PROPERTY bogKeyFilterOverloadToolValue : BOOL
GET
                    bogKeyFilterOverloadToolValue := bogKeyFilterOverload.Value;

                  
END_GET
SET
                    bogKeyFilterOverload.Value := bogKeyFilterOverloadToolValue;

                  
END_SET
END_PROPERTY

PROPERTY bogKeyNextModeToolValue : BOOL
GET
                    bogKeyNextModeToolValue := bogKeyNextMode.Value;

                  
END_GET
SET
                    bogKeyNextMode.Value := bogKeyNextModeToolValue;

                  
END_SET
END_PROPERTY

PROPERTY bogKeyPrevModeToolValue : BOOL
GET
                    bogKeyPrevModeToolValue := bogKeyPrevMode.Value;

                  
END_GET
SET
                    bogKeyPrevMode.Value := bogKeyPrevModeToolValue;

                  
END_SET
END_PROPERTY

PROPERTY bogKeySignalDangerToolValue : BOOL
GET
                    bogKeySignalDangerToolValue := bogKeySignalDanger.Value;

                  
END_GET
SET
                    bogKeySignalDanger.Value := bogKeySignalDangerToolValue;

                  
END_SET
END_PROPERTY

PROPERTY bogKeyFlashLightONToolValue : BOOL
GET
                    bogKeyFlashLightONToolValue := bogKeyFlashLightON.Value;

                  
END_GET
SET
                    bogKeyFlashLightON.Value := bogKeyFlashLightONToolValue;

                  
END_SET
END_PROPERTY

PROPERTY bogKeyCalibMastMinToolValue : BOOL
GET
                    bogKeyCalibMastMinToolValue := bogKeyCalibMastMin.Value;

                  
END_GET
SET
                    bogKeyCalibMastMin.Value := bogKeyCalibMastMinToolValue;

                  
END_SET
END_PROPERTY

PROPERTY bogKeyCalibMastMaxToolValue : BOOL
GET
                    bogKeyCalibMastMaxToolValue := bogKeyCalibMastMax.Value;

                  
END_GET
SET
                    bogKeyCalibMastMax.Value := bogKeyCalibMastMaxToolValue;

                  
END_SET
END_PROPERTY

PROPERTY bogKeyCalibMastValidToolValue : BOOL
GET
                    bogKeyCalibMastValidToolValue := bogKeyCalibMastValid.Value;

                  
END_GET
SET
                    bogKeyCalibMastValid.Value := bogKeyCalibMastValidToolValue;

                  
END_SET
END_PROPERTY

PROPERTY bogKeyGeneratorActivateToolValue : BOOL
GET
                    bogKeyGeneratorActivateToolValue := bogKeyGeneratorActivate.Value;

                  
END_GET
SET
                    bogKeyGeneratorActivate.Value := bogKeyGeneratorActivateToolValue;

                  
END_SET
END_PROPERTY

PROPERTY bogKeyWhiteLights15746ToolValue : BOOL
GET
                    bogKeyWhiteLights15746ToolValue := bogKeyWhiteLights15746.Value;

                  
END_GET
SET
                    bogKeyWhiteLights15746.Value := bogKeyWhiteLights15746ToolValue;

                  
END_SET
END_PROPERTY

PROPERTY bogFixe2ndParkBrakeSelectToolValue : BOOL
GET
                    bogFixe2ndParkBrakeSelectToolValue := bogFixe2ndParkBrakeSelect.Value;

                  
END_GET
SET
                    bogFixe2ndParkBrakeSelect.Value := bogFixe2ndParkBrakeSelectToolValue;

                  
END_SET
END_PROPERTY

PROPERTY bogOsci2ndParkBrakeSelectToolValue : BOOL
GET
                    bogOsci2ndParkBrakeSelectToolValue := bogOsci2ndParkBrakeSelect.Value;

                  
END_GET
SET
                    bogOsci2ndParkBrakeSelect.Value := bogOsci2ndParkBrakeSelectToolValue;

                  
END_SET
END_PROPERTY

PROPERTY bogKeyRazControllerToolValue : BOOL
GET
                    bogKeyRazControllerToolValue := bogKeyRazController.Value;

                  
END_GET
SET
                    bogKeyRazController.Value := bogKeyRazControllerToolValue;

                  
END_SET
END_PROPERTY

METHOD InitializeCanSignals
                  bogLoginStatus.AppScalingDivisor :=1;
bogLoginStatus.AppScalingMultiplier :=1;
bogLoginStatus.AppScalingOffset :=0;
bogLoginStatus.AppUnit :="[-]";
bogLoginStatus.CanDefault :=0;
bogLoginStatus.CanInit :=0;
bogLoginStatus.CanMax :=1;
bogLoginStatus.CanMin :=0;
bogLoginStatus.CanUnit :="";
bogLoginStatus.Description :="User Log in Status (1=log in)";
bogLoginStatus.ErrorReaction := eErrorReaction.ERSIG_DFLT;
bogLoginStatus.ReceiverAdress :=1;
bogLoginStatus.ToolScalingDivisor :=1;
bogLoginStatus.ToolScalingMultiplier :=1;
bogLoginStatus.ToolScalingOffset :=0;
bogLoginStatus.ToolUnit :="";

bogButtonCalibTurretEncoder.AppScalingDivisor :=1;
bogButtonCalibTurretEncoder.AppScalingMultiplier :=1;
bogButtonCalibTurretEncoder.AppScalingOffset :=0;
bogButtonCalibTurretEncoder.AppUnit :="[-]";
bogButtonCalibTurretEncoder.CanDefault :=0;
bogButtonCalibTurretEncoder.CanInit :=0;
bogButtonCalibTurretEncoder.CanMax :=1;
bogButtonCalibTurretEncoder.CanMin :=0;
bogButtonCalibTurretEncoder.CanUnit :="";
bogButtonCalibTurretEncoder.Description :="Button for the calibration of the turret encoder is pressed";
bogButtonCalibTurretEncoder.ErrorReaction := eErrorReaction.ERSIG_DFLT;
bogButtonCalibTurretEncoder.ReceiverAdress :=1;
bogButtonCalibTurretEncoder.ToolScalingDivisor :=1;
bogButtonCalibTurretEncoder.ToolScalingMultiplier :=1;
bogButtonCalibTurretEncoder.ToolScalingOffset :=0;
bogButtonCalibTurretEncoder.ToolUnit :="";

bogButtonCalibMinMastMeasure.AppScalingDivisor :=1;
bogButtonCalibMinMastMeasure.AppScalingMultiplier :=1;
bogButtonCalibMinMastMeasure.AppScalingOffset :=0;
bogButtonCalibMinMastMeasure.AppUnit :="[-]";
bogButtonCalibMinMastMeasure.CanDefault :=0;
bogButtonCalibMinMastMeasure.CanInit :=0;
bogButtonCalibMinMastMeasure.CanMax :=1;
bogButtonCalibMinMastMeasure.CanMin :=0;
bogButtonCalibMinMastMeasure.CanUnit :="";
bogButtonCalibMinMastMeasure.Description :="Button for the calibration of min position mast measure encodeur  is pressed";
bogButtonCalibMinMastMeasure.ErrorReaction := eErrorReaction.ERSIG_DFLT;
bogButtonCalibMinMastMeasure.ReceiverAdress :=1;
bogButtonCalibMinMastMeasure.ToolScalingDivisor :=1;
bogButtonCalibMinMastMeasure.ToolScalingMultiplier :=1;
bogButtonCalibMinMastMeasure.ToolScalingOffset :=0;
bogButtonCalibMinMastMeasure.ToolUnit :="";

bogButtonCalibMaxMastMeasure.AppScalingDivisor :=1;
bogButtonCalibMaxMastMeasure.AppScalingMultiplier :=1;
bogButtonCalibMaxMastMeasure.AppScalingOffset :=0;
bogButtonCalibMaxMastMeasure.AppUnit :="[-]";
bogButtonCalibMaxMastMeasure.CanDefault :=0;
bogButtonCalibMaxMastMeasure.CanInit :=0;
bogButtonCalibMaxMastMeasure.CanMax :=1;
bogButtonCalibMaxMastMeasure.CanMin :=0;
bogButtonCalibMaxMastMeasure.CanUnit :="";
bogButtonCalibMaxMastMeasure.Description :="Button for the calibration of max position mast measure encodeur  is pressed";
bogButtonCalibMaxMastMeasure.ErrorReaction := eErrorReaction.ERSIG_DFLT;
bogButtonCalibMaxMastMeasure.ReceiverAdress :=1;
bogButtonCalibMaxMastMeasure.ToolScalingDivisor :=1;
bogButtonCalibMaxMastMeasure.ToolScalingMultiplier :=1;
bogButtonCalibMaxMastMeasure.ToolScalingOffset :=0;
bogButtonCalibMaxMastMeasure.ToolUnit :="";

boSavePosEncodeurMastButton.AppScalingDivisor :=1;
boSavePosEncodeurMastButton.AppScalingMultiplier :=1;
boSavePosEncodeurMastButton.AppScalingOffset :=0;
boSavePosEncodeurMastButton.AppUnit :="[-]";
boSavePosEncodeurMastButton.CanDefault :=0;
boSavePosEncodeurMastButton.CanInit :=0;
boSavePosEncodeurMastButton.CanMax :=1;
boSavePosEncodeurMastButton.CanMin :=0;
boSavePosEncodeurMastButton.CanUnit :="";
boSavePosEncodeurMastButton.Description :="Button for save min and max value of encodeur mast measure";
boSavePosEncodeurMastButton.ErrorReaction := eErrorReaction.ERSIG_DFLT;
boSavePosEncodeurMastButton.ReceiverAdress :=1;
boSavePosEncodeurMastButton.ToolScalingDivisor :=1;
boSavePosEncodeurMastButton.ToolScalingMultiplier :=1;
boSavePosEncodeurMastButton.ToolScalingOffset :=0;
boSavePosEncodeurMastButton.ToolUnit :="";

bogActivateMeasuringMast.AppScalingDivisor :=1;
bogActivateMeasuringMast.AppScalingMultiplier :=1;
bogActivateMeasuringMast.AppScalingOffset :=0;
bogActivateMeasuringMast.AppUnit :="[-]";
bogActivateMeasuringMast.CanDefault :=0;
bogActivateMeasuringMast.CanInit :=0;
bogActivateMeasuringMast.CanMax :=1;
bogActivateMeasuringMast.CanMin :=0;
bogActivateMeasuringMast.CanUnit :="";
bogActivateMeasuringMast.Description :="Activate mast measure function";
bogActivateMeasuringMast.ErrorReaction := eErrorReaction.ERSIG_DFLT;
bogActivateMeasuringMast.ReceiverAdress :=1;
bogActivateMeasuringMast.ToolScalingDivisor :=1;
bogActivateMeasuringMast.ToolScalingMultiplier :=1;
bogActivateMeasuringMast.ToolScalingOffset :=0;
bogActivateMeasuringMast.ToolUnit :="";

boRazDistanceTraveledMastMeasure.AppScalingDivisor :=1;
boRazDistanceTraveledMastMeasure.AppScalingMultiplier :=1;
boRazDistanceTraveledMastMeasure.AppScalingOffset :=0;
boRazDistanceTraveledMastMeasure.AppUnit :="[-]";
boRazDistanceTraveledMastMeasure.CanDefault :=0;
boRazDistanceTraveledMastMeasure.CanInit :=0;
boRazDistanceTraveledMastMeasure.CanMax :=1;
boRazDistanceTraveledMastMeasure.CanMin :=0;
boRazDistanceTraveledMastMeasure.CanUnit :="";
boRazDistanceTraveledMastMeasure.Description :="Raz distance translation traveled with mast measure unfolded";
boRazDistanceTraveledMastMeasure.ErrorReaction := eErrorReaction.ERSIG_DFLT;
boRazDistanceTraveledMastMeasure.ReceiverAdress :=1;
boRazDistanceTraveledMastMeasure.ToolScalingDivisor :=1;
boRazDistanceTraveledMastMeasure.ToolScalingMultiplier :=1;
boRazDistanceTraveledMastMeasure.ToolScalingOffset :=0;
boRazDistanceTraveledMastMeasure.ToolUnit :="";

bogOffTrackTestBrakeActivated.AppScalingDivisor :=1;
bogOffTrackTestBrakeActivated.AppScalingMultiplier :=1;
bogOffTrackTestBrakeActivated.AppScalingOffset :=0;
bogOffTrackTestBrakeActivated.AppUnit :="[-]";
bogOffTrackTestBrakeActivated.CanDefault :=0;
bogOffTrackTestBrakeActivated.CanInit :=0;
bogOffTrackTestBrakeActivated.CanMax :=1;
bogOffTrackTestBrakeActivated.CanMin :=0;
bogOffTrackTestBrakeActivated.CanUnit :="";
bogOffTrackTestBrakeActivated.Description :="Status of off track variable on test brake page";
bogOffTrackTestBrakeActivated.ErrorReaction := eErrorReaction.ERSIG_DFLT;
bogOffTrackTestBrakeActivated.ReceiverAdress :=1;
bogOffTrackTestBrakeActivated.ToolScalingDivisor :=1;
bogOffTrackTestBrakeActivated.ToolScalingMultiplier :=1;
bogOffTrackTestBrakeActivated.ToolScalingOffset :=0;
bogOffTrackTestBrakeActivated.ToolUnit :="";

bogOffTrackRunInBrakeActivated.AppScalingDivisor :=1;
bogOffTrackRunInBrakeActivated.AppScalingMultiplier :=1;
bogOffTrackRunInBrakeActivated.AppScalingOffset :=0;
bogOffTrackRunInBrakeActivated.AppUnit :="[-]";
bogOffTrackRunInBrakeActivated.CanDefault :=0;
bogOffTrackRunInBrakeActivated.CanInit :=0;
bogOffTrackRunInBrakeActivated.CanMax :=1;
bogOffTrackRunInBrakeActivated.CanMin :=0;
bogOffTrackRunInBrakeActivated.CanUnit :="";
bogOffTrackRunInBrakeActivated.Description :="Status of off track variable on run in process page";
bogOffTrackRunInBrakeActivated.ErrorReaction := eErrorReaction.ERSIG_DFLT;
bogOffTrackRunInBrakeActivated.ReceiverAdress :=1;
bogOffTrackRunInBrakeActivated.ToolScalingDivisor :=1;
bogOffTrackRunInBrakeActivated.ToolScalingMultiplier :=1;
bogOffTrackRunInBrakeActivated.ToolScalingOffset :=0;
bogOffTrackRunInBrakeActivated.ToolUnit :="";

bogOsciServiceBrakeSelect.AppScalingDivisor :=1;
bogOsciServiceBrakeSelect.AppScalingMultiplier :=1;
bogOsciServiceBrakeSelect.AppScalingOffset :=0;
bogOsciServiceBrakeSelect.AppUnit :="[-]";
bogOsciServiceBrakeSelect.CanDefault :=0;
bogOsciServiceBrakeSelect.CanInit :=0;
bogOsciServiceBrakeSelect.CanMax :=1;
bogOsciServiceBrakeSelect.CanMin :=0;
bogOsciServiceBrakeSelect.CanUnit :="";
bogOsciServiceBrakeSelect.Description :="Request status of osci service test brake";
bogOsciServiceBrakeSelect.ErrorReaction := eErrorReaction.ERSIG_DFLT;
bogOsciServiceBrakeSelect.ReceiverAdress :=1;
bogOsciServiceBrakeSelect.ToolScalingDivisor :=1;
bogOsciServiceBrakeSelect.ToolScalingMultiplier :=1;
bogOsciServiceBrakeSelect.ToolScalingOffset :=0;
bogOsciServiceBrakeSelect.ToolUnit :="";

bogFixedServiceBrakeSelect.AppScalingDivisor :=1;
bogFixedServiceBrakeSelect.AppScalingMultiplier :=1;
bogFixedServiceBrakeSelect.AppScalingOffset :=0;
bogFixedServiceBrakeSelect.AppUnit :="[-]";
bogFixedServiceBrakeSelect.CanDefault :=0;
bogFixedServiceBrakeSelect.CanInit :=0;
bogFixedServiceBrakeSelect.CanMax :=1;
bogFixedServiceBrakeSelect.CanMin :=0;
bogFixedServiceBrakeSelect.CanUnit :="";
bogFixedServiceBrakeSelect.Description :="Request status of fixed service test brake";
bogFixedServiceBrakeSelect.ErrorReaction := eErrorReaction.ERSIG_DFLT;
bogFixedServiceBrakeSelect.ReceiverAdress :=1;
bogFixedServiceBrakeSelect.ToolScalingDivisor :=1;
bogFixedServiceBrakeSelect.ToolScalingMultiplier :=1;
bogFixedServiceBrakeSelect.ToolScalingOffset :=0;
bogFixedServiceBrakeSelect.ToolUnit :="";

bogBothServiceBrakeSelect.AppScalingDivisor :=1;
bogBothServiceBrakeSelect.AppScalingMultiplier :=1;
bogBothServiceBrakeSelect.AppScalingOffset :=0;
bogBothServiceBrakeSelect.AppUnit :="[-]";
bogBothServiceBrakeSelect.CanDefault :=0;
bogBothServiceBrakeSelect.CanInit :=0;
bogBothServiceBrakeSelect.CanMax :=1;
bogBothServiceBrakeSelect.CanMin :=0;
bogBothServiceBrakeSelect.CanUnit :="";
bogBothServiceBrakeSelect.Description :="Request status of both service test brake";
bogBothServiceBrakeSelect.ErrorReaction := eErrorReaction.ERSIG_DFLT;
bogBothServiceBrakeSelect.ReceiverAdress :=1;
bogBothServiceBrakeSelect.ToolScalingDivisor :=1;
bogBothServiceBrakeSelect.ToolScalingMultiplier :=1;
bogBothServiceBrakeSelect.ToolScalingOffset :=0;
bogBothServiceBrakeSelect.ToolUnit :="";

bogOsciParkBrakeSelect.AppScalingDivisor :=1;
bogOsciParkBrakeSelect.AppScalingMultiplier :=1;
bogOsciParkBrakeSelect.AppScalingOffset :=0;
bogOsciParkBrakeSelect.AppUnit :="[-]";
bogOsciParkBrakeSelect.CanDefault :=0;
bogOsciParkBrakeSelect.CanInit :=0;
bogOsciParkBrakeSelect.CanMax :=1;
bogOsciParkBrakeSelect.CanMin :=0;
bogOsciParkBrakeSelect.CanUnit :="";
bogOsciParkBrakeSelect.Description :="Request status of osci park test brake";
bogOsciParkBrakeSelect.ErrorReaction := eErrorReaction.ERSIG_DFLT;
bogOsciParkBrakeSelect.ReceiverAdress :=1;
bogOsciParkBrakeSelect.ToolScalingDivisor :=1;
bogOsciParkBrakeSelect.ToolScalingMultiplier :=1;
bogOsciParkBrakeSelect.ToolScalingOffset :=0;
bogOsciParkBrakeSelect.ToolUnit :="";

bogFixedParkBrakeSelect.AppScalingDivisor :=1;
bogFixedParkBrakeSelect.AppScalingMultiplier :=1;
bogFixedParkBrakeSelect.AppScalingOffset :=0;
bogFixedParkBrakeSelect.AppUnit :="[-]";
bogFixedParkBrakeSelect.CanDefault :=0;
bogFixedParkBrakeSelect.CanInit :=0;
bogFixedParkBrakeSelect.CanMax :=1;
bogFixedParkBrakeSelect.CanMin :=0;
bogFixedParkBrakeSelect.CanUnit :="";
bogFixedParkBrakeSelect.Description :="Request status of fixed park test brake";
bogFixedParkBrakeSelect.ErrorReaction := eErrorReaction.ERSIG_DFLT;
bogFixedParkBrakeSelect.ReceiverAdress :=1;
bogFixedParkBrakeSelect.ToolScalingDivisor :=1;
bogFixedParkBrakeSelect.ToolScalingMultiplier :=1;
bogFixedParkBrakeSelect.ToolScalingOffset :=0;
bogFixedParkBrakeSelect.ToolUnit :="";

bogBothParkBrakeSelect.AppScalingDivisor :=1;
bogBothParkBrakeSelect.AppScalingMultiplier :=1;
bogBothParkBrakeSelect.AppScalingOffset :=0;
bogBothParkBrakeSelect.AppUnit :="[-]";
bogBothParkBrakeSelect.CanDefault :=0;
bogBothParkBrakeSelect.CanInit :=0;
bogBothParkBrakeSelect.CanMax :=1;
bogBothParkBrakeSelect.CanMin :=0;
bogBothParkBrakeSelect.CanUnit :="";
bogBothParkBrakeSelect.Description :="Request status of both park test brake";
bogBothParkBrakeSelect.ErrorReaction := eErrorReaction.ERSIG_DFLT;
bogBothParkBrakeSelect.ReceiverAdress :=1;
bogBothParkBrakeSelect.ToolScalingDivisor :=1;
bogBothParkBrakeSelect.ToolScalingMultiplier :=1;
bogBothParkBrakeSelect.ToolScalingOffset :=0;
bogBothParkBrakeSelect.ToolUnit :="";

bogOsciServiceRunInBrakeSelect.AppScalingDivisor :=1;
bogOsciServiceRunInBrakeSelect.AppScalingMultiplier :=1;
bogOsciServiceRunInBrakeSelect.AppScalingOffset :=0;
bogOsciServiceRunInBrakeSelect.AppUnit :="[-]";
bogOsciServiceRunInBrakeSelect.CanDefault :=0;
bogOsciServiceRunInBrakeSelect.CanInit :=0;
bogOsciServiceRunInBrakeSelect.CanMax :=1;
bogOsciServiceRunInBrakeSelect.CanMin :=0;
bogOsciServiceRunInBrakeSelect.CanUnit :="";
bogOsciServiceRunInBrakeSelect.Description :="Request status of osci service run in brake";
bogOsciServiceRunInBrakeSelect.ErrorReaction := eErrorReaction.ERSIG_DFLT;
bogOsciServiceRunInBrakeSelect.ReceiverAdress :=1;
bogOsciServiceRunInBrakeSelect.ToolScalingDivisor :=1;
bogOsciServiceRunInBrakeSelect.ToolScalingMultiplier :=1;
bogOsciServiceRunInBrakeSelect.ToolScalingOffset :=0;
bogOsciServiceRunInBrakeSelect.ToolUnit :="";

bogFixedServiceRunInBrakeSelect.AppScalingDivisor :=1;
bogFixedServiceRunInBrakeSelect.AppScalingMultiplier :=1;
bogFixedServiceRunInBrakeSelect.AppScalingOffset :=0;
bogFixedServiceRunInBrakeSelect.AppUnit :="[-]";
bogFixedServiceRunInBrakeSelect.CanDefault :=0;
bogFixedServiceRunInBrakeSelect.CanInit :=0;
bogFixedServiceRunInBrakeSelect.CanMax :=1;
bogFixedServiceRunInBrakeSelect.CanMin :=0;
bogFixedServiceRunInBrakeSelect.CanUnit :="";
bogFixedServiceRunInBrakeSelect.Description :="Request status of fixed service run in test brake";
bogFixedServiceRunInBrakeSelect.ErrorReaction := eErrorReaction.ERSIG_DFLT;
bogFixedServiceRunInBrakeSelect.ReceiverAdress :=1;
bogFixedServiceRunInBrakeSelect.ToolScalingDivisor :=1;
bogFixedServiceRunInBrakeSelect.ToolScalingMultiplier :=1;
bogFixedServiceRunInBrakeSelect.ToolScalingOffset :=0;
bogFixedServiceRunInBrakeSelect.ToolUnit :="";

bogBothServiceRunInBrakeSelect.AppScalingDivisor :=1;
bogBothServiceRunInBrakeSelect.AppScalingMultiplier :=1;
bogBothServiceRunInBrakeSelect.AppScalingOffset :=0;
bogBothServiceRunInBrakeSelect.AppUnit :="[-]";
bogBothServiceRunInBrakeSelect.CanDefault :=0;
bogBothServiceRunInBrakeSelect.CanInit :=0;
bogBothServiceRunInBrakeSelect.CanMax :=1;
bogBothServiceRunInBrakeSelect.CanMin :=0;
bogBothServiceRunInBrakeSelect.CanUnit :="";
bogBothServiceRunInBrakeSelect.Description :="Request status of both service run in test brake";
bogBothServiceRunInBrakeSelect.ErrorReaction := eErrorReaction.ERSIG_DFLT;
bogBothServiceRunInBrakeSelect.ReceiverAdress :=1;
bogBothServiceRunInBrakeSelect.ToolScalingDivisor :=1;
bogBothServiceRunInBrakeSelect.ToolScalingMultiplier :=1;
bogBothServiceRunInBrakeSelect.ToolScalingOffset :=0;
bogBothServiceRunInBrakeSelect.ToolUnit :="";

bogTestBrakePageActive.AppScalingDivisor :=1;
bogTestBrakePageActive.AppScalingMultiplier :=1;
bogTestBrakePageActive.AppScalingOffset :=0;
bogTestBrakePageActive.AppUnit :="[-]";
bogTestBrakePageActive.CanDefault :=0;
bogTestBrakePageActive.CanInit :=0;
bogTestBrakePageActive.CanMax :=1;
bogTestBrakePageActive.CanMin :=0;
bogTestBrakePageActive.CanUnit :="";
bogTestBrakePageActive.Description :="Flag when user is on test brake page";
bogTestBrakePageActive.ErrorReaction := eErrorReaction.ERSIG_DFLT;
bogTestBrakePageActive.ReceiverAdress :=1;
bogTestBrakePageActive.ToolScalingDivisor :=1;
bogTestBrakePageActive.ToolScalingMultiplier :=1;
bogTestBrakePageActive.ToolScalingOffset :=0;
bogTestBrakePageActive.ToolUnit :="";

bogBreakInBrakePageActive.AppScalingDivisor :=1;
bogBreakInBrakePageActive.AppScalingMultiplier :=1;
bogBreakInBrakePageActive.AppScalingOffset :=0;
bogBreakInBrakePageActive.AppUnit :="[-]";
bogBreakInBrakePageActive.CanDefault :=0;
bogBreakInBrakePageActive.CanInit :=0;
bogBreakInBrakePageActive.CanMax :=1;
bogBreakInBrakePageActive.CanMin :=0;
bogBreakInBrakePageActive.CanUnit :="";
bogBreakInBrakePageActive.Description :="Flag when user is on break in brake page";
bogBreakInBrakePageActive.ErrorReaction := eErrorReaction.ERSIG_DFLT;
bogBreakInBrakePageActive.ReceiverAdress :=1;
bogBreakInBrakePageActive.ToolScalingDivisor :=1;
bogBreakInBrakePageActive.ToolScalingMultiplier :=1;
bogBreakInBrakePageActive.ToolScalingOffset :=0;
bogBreakInBrakePageActive.ToolUnit :="";

bogSerialNumber.AppScalingDivisor :=1;
bogSerialNumber.AppScalingMultiplier :=1;
bogSerialNumber.AppScalingOffset :=0;
bogSerialNumber.AppUnit :="[-]";
bogSerialNumber.CanDefault :=0;
bogSerialNumber.CanInit :=0;
bogSerialNumber.CanMax :=1;
bogSerialNumber.CanMin :=0;
bogSerialNumber.CanUnit :="";
bogSerialNumber.Description :="Machine Serial Number";
bogSerialNumber.ErrorReaction := eErrorReaction.ERSIG_DFLT;
bogSerialNumber.ReceiverAdress :=1;
bogSerialNumber.ToolScalingDivisor :=1;
bogSerialNumber.ToolScalingMultiplier :=1;
bogSerialNumber.ToolScalingOffset :=0;
bogSerialNumber.ToolUnit :="";

bogBPBasketValidate.AppScalingDivisor :=1;
bogBPBasketValidate.AppScalingMultiplier :=1;
bogBPBasketValidate.AppScalingOffset :=0;
bogBPBasketValidate.AppUnit :="[-]";
bogBPBasketValidate.CanDefault :=0;
bogBPBasketValidate.CanInit :=0;
bogBPBasketValidate.CanMax :=1;
bogBPBasketValidate.CanMin :=0;
bogBPBasketValidate.CanUnit :="";
bogBPBasketValidate.Description :="Basket Panel Validate";
bogBPBasketValidate.ErrorReaction := eErrorReaction.ERSIG_DFLT;
bogBPBasketValidate.ReceiverAdress :=1;
bogBPBasketValidate.ToolScalingDivisor :=1;
bogBPBasketValidate.ToolScalingMultiplier :=1;
bogBPBasketValidate.ToolScalingOffset :=0;
bogBPBasketValidate.ToolUnit :="";

bogKeyFilterOverload.AppScalingDivisor :=1;
bogKeyFilterOverload.AppScalingMultiplier :=1;
bogKeyFilterOverload.AppScalingOffset :=0;
bogKeyFilterOverload.AppUnit :="[-]";
bogKeyFilterOverload.CanDefault :=0;
bogKeyFilterOverload.CanInit :=0;
bogKeyFilterOverload.CanMax :=1;
bogKeyFilterOverload.CanMin :=0;
bogKeyFilterOverload.CanUnit :="";
bogKeyFilterOverload.Description :="Overload Filter Key";
bogKeyFilterOverload.ErrorReaction := eErrorReaction.ERSIG_DFLT;
bogKeyFilterOverload.ReceiverAdress :=1;
bogKeyFilterOverload.ToolScalingDivisor :=1;
bogKeyFilterOverload.ToolScalingMultiplier :=1;
bogKeyFilterOverload.ToolScalingOffset :=0;
bogKeyFilterOverload.ToolUnit :="";

bogKeyNextMode.AppScalingDivisor :=1;
bogKeyNextMode.AppScalingMultiplier :=1;
bogKeyNextMode.AppScalingOffset :=0;
bogKeyNextMode.AppUnit :="[-]";
bogKeyNextMode.CanDefault :=0;
bogKeyNextMode.CanInit :=0;
bogKeyNextMode.CanMax :=1;
bogKeyNextMode.CanMin :=0;
bogKeyNextMode.CanUnit :="";
bogKeyNextMode.Description :="Select next mode";
bogKeyNextMode.ErrorReaction := eErrorReaction.ERSIG_DFLT;
bogKeyNextMode.ReceiverAdress :=1;
bogKeyNextMode.ToolScalingDivisor :=1;
bogKeyNextMode.ToolScalingMultiplier :=1;
bogKeyNextMode.ToolScalingOffset :=0;
bogKeyNextMode.ToolUnit :="";

bogKeyPrevMode.AppScalingDivisor :=1;
bogKeyPrevMode.AppScalingMultiplier :=1;
bogKeyPrevMode.AppScalingOffset :=0;
bogKeyPrevMode.AppUnit :="[-]";
bogKeyPrevMode.CanDefault :=0;
bogKeyPrevMode.CanInit :=0;
bogKeyPrevMode.CanMax :=1;
bogKeyPrevMode.CanMin :=0;
bogKeyPrevMode.CanUnit :="";
bogKeyPrevMode.Description :="Select Previous Mode";
bogKeyPrevMode.ErrorReaction := eErrorReaction.ERSIG_DFLT;
bogKeyPrevMode.ReceiverAdress :=1;
bogKeyPrevMode.ToolScalingDivisor :=1;
bogKeyPrevMode.ToolScalingMultiplier :=1;
bogKeyPrevMode.ToolScalingOffset :=0;
bogKeyPrevMode.ToolUnit :="";

bogKeySignalDanger.AppScalingDivisor :=1;
bogKeySignalDanger.AppScalingMultiplier :=1;
bogKeySignalDanger.AppScalingOffset :=0;
bogKeySignalDanger.AppUnit :="[-]";
bogKeySignalDanger.CanDefault :=0;
bogKeySignalDanger.CanInit :=0;
bogKeySignalDanger.CanMax :=1;
bogKeySignalDanger.CanMin :=0;
bogKeySignalDanger.CanUnit :="";
bogKeySignalDanger.Description :="Select Signal Danger Mode";
bogKeySignalDanger.ErrorReaction := eErrorReaction.ERSIG_DFLT;
bogKeySignalDanger.ReceiverAdress :=1;
bogKeySignalDanger.ToolScalingDivisor :=1;
bogKeySignalDanger.ToolScalingMultiplier :=1;
bogKeySignalDanger.ToolScalingOffset :=0;
bogKeySignalDanger.ToolUnit :="";

bogKeyFlashLightON.AppScalingDivisor :=1;
bogKeyFlashLightON.AppScalingMultiplier :=1;
bogKeyFlashLightON.AppScalingOffset :=0;
bogKeyFlashLightON.AppUnit :="[-]";
bogKeyFlashLightON.CanDefault :=0;
bogKeyFlashLightON.CanInit :=0;
bogKeyFlashLightON.CanMax :=1;
bogKeyFlashLightON.CanMin :=0;
bogKeyFlashLightON.CanUnit :="";
bogKeyFlashLightON.Description :="Force Flash Light ON";
bogKeyFlashLightON.ErrorReaction := eErrorReaction.ERSIG_DFLT;
bogKeyFlashLightON.ReceiverAdress :=1;
bogKeyFlashLightON.ToolScalingDivisor :=1;
bogKeyFlashLightON.ToolScalingMultiplier :=1;
bogKeyFlashLightON.ToolScalingOffset :=0;
bogKeyFlashLightON.ToolUnit :="";

bogKeyCalibMastMin.AppScalingDivisor :=1;
bogKeyCalibMastMin.AppScalingMultiplier :=1;
bogKeyCalibMastMin.AppScalingOffset :=0;
bogKeyCalibMastMin.AppUnit :="[-]";
bogKeyCalibMastMin.CanDefault :=0;
bogKeyCalibMastMin.CanInit :=0;
bogKeyCalibMastMin.CanMax :=1;
bogKeyCalibMastMin.CanMin :=0;
bogKeyCalibMastMin.CanUnit :="";
bogKeyCalibMastMin.Description :="Key Calibration Min";
bogKeyCalibMastMin.ErrorReaction := eErrorReaction.ERSIG_DFLT;
bogKeyCalibMastMin.ReceiverAdress :=1;
bogKeyCalibMastMin.ToolScalingDivisor :=1;
bogKeyCalibMastMin.ToolScalingMultiplier :=1;
bogKeyCalibMastMin.ToolScalingOffset :=0;
bogKeyCalibMastMin.ToolUnit :="";

bogKeyCalibMastMax.AppScalingDivisor :=1;
bogKeyCalibMastMax.AppScalingMultiplier :=1;
bogKeyCalibMastMax.AppScalingOffset :=0;
bogKeyCalibMastMax.AppUnit :="[-]";
bogKeyCalibMastMax.CanDefault :=0;
bogKeyCalibMastMax.CanInit :=0;
bogKeyCalibMastMax.CanMax :=1;
bogKeyCalibMastMax.CanMin :=0;
bogKeyCalibMastMax.CanUnit :="";
bogKeyCalibMastMax.Description :="Key Calibration Max";
bogKeyCalibMastMax.ErrorReaction := eErrorReaction.ERSIG_DFLT;
bogKeyCalibMastMax.ReceiverAdress :=1;
bogKeyCalibMastMax.ToolScalingDivisor :=1;
bogKeyCalibMastMax.ToolScalingMultiplier :=1;
bogKeyCalibMastMax.ToolScalingOffset :=0;
bogKeyCalibMastMax.ToolUnit :="";

bogKeyCalibMastValid.AppScalingDivisor :=1;
bogKeyCalibMastValid.AppScalingMultiplier :=1;
bogKeyCalibMastValid.AppScalingOffset :=0;
bogKeyCalibMastValid.AppUnit :="[-]";
bogKeyCalibMastValid.CanDefault :=0;
bogKeyCalibMastValid.CanInit :=0;
bogKeyCalibMastValid.CanMax :=1;
bogKeyCalibMastValid.CanMin :=0;
bogKeyCalibMastValid.CanUnit :="";
bogKeyCalibMastValid.Description :="Key Calibration Validation";
bogKeyCalibMastValid.ErrorReaction := eErrorReaction.ERSIG_DFLT;
bogKeyCalibMastValid.ReceiverAdress :=1;
bogKeyCalibMastValid.ToolScalingDivisor :=1;
bogKeyCalibMastValid.ToolScalingMultiplier :=1;
bogKeyCalibMastValid.ToolScalingOffset :=0;
bogKeyCalibMastValid.ToolUnit :="";

bogKeyGeneratorActivate.AppScalingDivisor :=1;
bogKeyGeneratorActivate.AppScalingMultiplier :=1;
bogKeyGeneratorActivate.AppScalingOffset :=0;
bogKeyGeneratorActivate.AppUnit :="[-]";
bogKeyGeneratorActivate.CanDefault :=0;
bogKeyGeneratorActivate.CanInit :=0;
bogKeyGeneratorActivate.CanMax :=1;
bogKeyGeneratorActivate.CanMin :=0;
bogKeyGeneratorActivate.CanUnit :="";
bogKeyGeneratorActivate.Description :="Key Generator Activation";
bogKeyGeneratorActivate.ErrorReaction := eErrorReaction.ERSIG_DFLT;
bogKeyGeneratorActivate.ReceiverAdress :=1;
bogKeyGeneratorActivate.ToolScalingDivisor :=1;
bogKeyGeneratorActivate.ToolScalingMultiplier :=1;
bogKeyGeneratorActivate.ToolScalingOffset :=0;
bogKeyGeneratorActivate.ToolUnit :="";

bogKeyWhiteLights15746.AppScalingDivisor :=1;
bogKeyWhiteLights15746.AppScalingMultiplier :=1;
bogKeyWhiteLights15746.AppScalingOffset :=0;
bogKeyWhiteLights15746.AppUnit :="[-]";
bogKeyWhiteLights15746.CanDefault :=0;
bogKeyWhiteLights15746.CanInit :=0;
bogKeyWhiteLights15746.CanMax :=1;
bogKeyWhiteLights15746.CanMin :=0;
bogKeyWhiteLights15746.CanUnit :="";
bogKeyWhiteLights15746.Description :="Key whiite lights 15746";
bogKeyWhiteLights15746.ErrorReaction := eErrorReaction.ERSIG_DFLT;
bogKeyWhiteLights15746.ReceiverAdress :=1;
bogKeyWhiteLights15746.ToolScalingDivisor :=1;
bogKeyWhiteLights15746.ToolScalingMultiplier :=1;
bogKeyWhiteLights15746.ToolScalingOffset :=0;
bogKeyWhiteLights15746.ToolUnit :="";

bogFixe2ndParkBrakeSelect.AppScalingDivisor :=1;
bogFixe2ndParkBrakeSelect.AppScalingMultiplier :=1;
bogFixe2ndParkBrakeSelect.AppScalingOffset :=0;
bogFixe2ndParkBrakeSelect.AppUnit :="[-]";
bogFixe2ndParkBrakeSelect.CanDefault :=0;
bogFixe2ndParkBrakeSelect.CanInit :=0;
bogFixe2ndParkBrakeSelect.CanMax :=1;
bogFixe2ndParkBrakeSelect.CanMin :=0;
bogFixe2ndParkBrakeSelect.CanUnit :="";
bogFixe2ndParkBrakeSelect.Description :="Fixe 2nd Park Brake Select";
bogFixe2ndParkBrakeSelect.ErrorReaction := eErrorReaction.ERSIG_DFLT;
bogFixe2ndParkBrakeSelect.ReceiverAdress :=1;
bogFixe2ndParkBrakeSelect.ToolScalingDivisor :=1;
bogFixe2ndParkBrakeSelect.ToolScalingMultiplier :=1;
bogFixe2ndParkBrakeSelect.ToolScalingOffset :=0;
bogFixe2ndParkBrakeSelect.ToolUnit :="";

bogOsci2ndParkBrakeSelect.AppScalingDivisor :=1;
bogOsci2ndParkBrakeSelect.AppScalingMultiplier :=1;
bogOsci2ndParkBrakeSelect.AppScalingOffset :=0;
bogOsci2ndParkBrakeSelect.AppUnit :="[-]";
bogOsci2ndParkBrakeSelect.CanDefault :=0;
bogOsci2ndParkBrakeSelect.CanInit :=0;
bogOsci2ndParkBrakeSelect.CanMax :=1;
bogOsci2ndParkBrakeSelect.CanMin :=0;
bogOsci2ndParkBrakeSelect.CanUnit :="";
bogOsci2ndParkBrakeSelect.Description :="Osci 2nd Park Brake Select";
bogOsci2ndParkBrakeSelect.ErrorReaction := eErrorReaction.ERSIG_DFLT;
bogOsci2ndParkBrakeSelect.ReceiverAdress :=1;
bogOsci2ndParkBrakeSelect.ToolScalingDivisor :=1;
bogOsci2ndParkBrakeSelect.ToolScalingMultiplier :=1;
bogOsci2ndParkBrakeSelect.ToolScalingOffset :=0;
bogOsci2ndParkBrakeSelect.ToolUnit :="";

bogKeyRazController.AppScalingDivisor :=1;
bogKeyRazController.AppScalingMultiplier :=1;
bogKeyRazController.AppScalingOffset :=0;
bogKeyRazController.AppUnit :="[-]";
bogKeyRazController.CanDefault :=0;
bogKeyRazController.CanInit :=0;
bogKeyRazController.CanMax :=1;
bogKeyRazController.CanMin :=0;
bogKeyRazController.CanUnit :="";
bogKeyRazController.Description :="new signal";
bogKeyRazController.ErrorReaction := eErrorReaction.ERSIG_DFLT;
bogKeyRazController.ReceiverAdress :=1;
bogKeyRazController.ToolScalingDivisor :=1;
bogKeyRazController.ToolScalingMultiplier :=1;
bogKeyRazController.ToolScalingOffset :=0;
bogKeyRazController.ToolUnit :="";


                
END_METHOD

METHOD InvalidateNonVisuals
                  //Detect if there were data changes in this cycle and set the internal var
fDataChanged := bogLoginStatus.Changed OR
	bogButtonCalibTurretEncoder.Changed OR
	bogButtonCalibMinMastMeasure.Changed OR
	bogButtonCalibMaxMastMeasure.Changed OR
	boSavePosEncodeurMastButton.Changed OR
	bogActivateMeasuringMast.Changed OR
	boRazDistanceTraveledMastMeasure.Changed OR
	bogOffTrackTestBrakeActivated.Changed OR
	bogOffTrackRunInBrakeActivated.Changed OR
	bogOsciServiceBrakeSelect.Changed OR
	bogFixedServiceBrakeSelect.Changed OR
	bogBothServiceBrakeSelect.Changed OR
	bogOsciParkBrakeSelect.Changed OR
	bogFixedParkBrakeSelect.Changed OR
	bogBothParkBrakeSelect.Changed OR
	bogOsciServiceRunInBrakeSelect.Changed OR
	bogFixedServiceRunInBrakeSelect.Changed OR
	bogBothServiceRunInBrakeSelect.Changed OR
	bogTestBrakePageActive.Changed OR
	bogBreakInBrakePageActive.Changed OR
	bogSerialNumber.Changed OR
	bogBPBasketValidate.Changed OR
	bogKeyFilterOverload.Changed OR
	bogKeyNextMode.Changed OR
	bogKeyPrevMode.Changed OR
	bogKeySignalDanger.Changed OR
	bogKeyFlashLightON.Changed OR
	bogKeyCalibMastMin.Changed OR
	bogKeyCalibMastMax.Changed OR
	bogKeyCalibMastValid.Changed OR
	bogKeyGeneratorActivate.Changed OR
	bogKeyWhiteLights15746.Changed OR
	bogFixe2ndParkBrakeSelect.Changed OR
	bogOsci2ndParkBrakeSelect.Changed OR
	bogKeyRazController.Changed;
SUPER^.InvalidateNonVisuals();
IF fSendMessage THEN
	_sendMessage();
END_IF

                
END_METHOD
END_FUNCTION_BLOCK

FUNCTION_BLOCK Msg8C1SendToOpusMessageClass EXTENDS CanReceiveMessageClass
  VAR_INPUT
    u8gTTC510Version_Major : UInt8CanSignalClass;
    u8gTTC510Version_Minor : UInt8CanSignalClass;
    u8gTTC510Version_Patch : UInt8CanSignalClass;
    u8gTTC510Version_Custom : UInt8CanSignalClass;
    u8gTTC48XSVersion_Major : UInt8CanSignalClass;
    u8gTTC48XSVersion_Minor : UInt8CanSignalClass;
    u8gTTC48XSVersion_Patch : UInt8CanSignalClass;
    u8gTTC48XSVersion_Custom : UInt8CanSignalClass;
    Counter : UInt32CanSignalClass;
  END_VAR

            
          

METHOD SetData
  VAR_INPUT
    CanMsgPointer : POINTER TO CanMessageClass;
  END_VAR
                  IF IsValidPointer(canMsgPointer,'SetData') THEN
	SUPER^.SetData(CanMsgPointer);
	//Set the new data
	u8gTTC510Version_Major.Value := canMsgPointer^.GetUint8(0);
	u8gTTC510Version_Minor.Value := canMsgPointer^.GetUint8(8);
	u8gTTC510Version_Patch.Value := canMsgPointer^.GetUint8(16);
	u8gTTC510Version_Custom.Value := canMsgPointer^.GetUint8(24);
	u8gTTC48XSVersion_Major.Value := canMsgPointer^.GetUint8(32);
	u8gTTC48XSVersion_Minor.Value := canMsgPointer^.GetUint8(40);
	u8gTTC48XSVersion_Patch.Value := canMsgPointer^.GetUint8(48);
	u8gTTC48XSVersion_Custom.Value := canMsgPointer^.GetUint8(56);
	//And increase the counter
	Counter.Value := CanMsgPointer^.Counter.Value;
END_IF

                
END_METHOD

PROPERTY u8gTTC510Version_MajorRawValue : USINT
GET
                    IF u8gTTC510Version_Major.AppScalingMultiplier = 0 THEN
	_MatchLog^.Error("Get u8gTTC510Version_MajorRawValue", "Division by Zero!");
	RETURN;
End_IF

u8gTTC510Version_MajorRawValue := TO_USINT((u8gTTC510Version_Major.Value - u8gTTC510Version_Major.AppScalingOffset) * u8gTTC510Version_Major.AppScalingDivisor / u8gTTC510Version_Major.AppScalingMultiplier);

                  
END_GET
END_PROPERTY

PROPERTY u8gTTC510Version_MinorRawValue : USINT
GET
                    IF u8gTTC510Version_Minor.AppScalingMultiplier = 0 THEN
	_MatchLog^.Error("Get u8gTTC510Version_MinorRawValue", "Division by Zero!");
	RETURN;
End_IF

u8gTTC510Version_MinorRawValue := TO_USINT((u8gTTC510Version_Minor.Value - u8gTTC510Version_Minor.AppScalingOffset) * u8gTTC510Version_Minor.AppScalingDivisor / u8gTTC510Version_Minor.AppScalingMultiplier);

                  
END_GET
END_PROPERTY

PROPERTY u8gTTC510Version_PatchRawValue : USINT
GET
                    IF u8gTTC510Version_Patch.AppScalingMultiplier = 0 THEN
	_MatchLog^.Error("Get u8gTTC510Version_PatchRawValue", "Division by Zero!");
	RETURN;
End_IF

u8gTTC510Version_PatchRawValue := TO_USINT((u8gTTC510Version_Patch.Value - u8gTTC510Version_Patch.AppScalingOffset) * u8gTTC510Version_Patch.AppScalingDivisor / u8gTTC510Version_Patch.AppScalingMultiplier);

                  
END_GET
END_PROPERTY

PROPERTY u8gTTC510Version_CustomRawValue : USINT
GET
                    IF u8gTTC510Version_Custom.AppScalingMultiplier = 0 THEN
	_MatchLog^.Error("Get u8gTTC510Version_CustomRawValue", "Division by Zero!");
	RETURN;
End_IF

u8gTTC510Version_CustomRawValue := TO_USINT((u8gTTC510Version_Custom.Value - u8gTTC510Version_Custom.AppScalingOffset) * u8gTTC510Version_Custom.AppScalingDivisor / u8gTTC510Version_Custom.AppScalingMultiplier);

                  
END_GET
END_PROPERTY

PROPERTY u8gTTC48XSVersion_MajorRawValue : USINT
GET
                    IF u8gTTC48XSVersion_Major.AppScalingMultiplier = 0 THEN
	_MatchLog^.Error("Get u8gTTC48XSVersion_MajorRawValue", "Division by Zero!");
	RETURN;
End_IF

u8gTTC48XSVersion_MajorRawValue := TO_USINT((u8gTTC48XSVersion_Major.Value - u8gTTC48XSVersion_Major.AppScalingOffset) * u8gTTC48XSVersion_Major.AppScalingDivisor / u8gTTC48XSVersion_Major.AppScalingMultiplier);

                  
END_GET
END_PROPERTY

PROPERTY u8gTTC48XSVersion_MinorRawValue : USINT
GET
                    IF u8gTTC48XSVersion_Minor.AppScalingMultiplier = 0 THEN
	_MatchLog^.Error("Get u8gTTC48XSVersion_MinorRawValue", "Division by Zero!");
	RETURN;
End_IF

u8gTTC48XSVersion_MinorRawValue := TO_USINT((u8gTTC48XSVersion_Minor.Value - u8gTTC48XSVersion_Minor.AppScalingOffset) * u8gTTC48XSVersion_Minor.AppScalingDivisor / u8gTTC48XSVersion_Minor.AppScalingMultiplier);

                  
END_GET
END_PROPERTY

PROPERTY u8gTTC48XSVersion_PatchRawValue : USINT
GET
                    IF u8gTTC48XSVersion_Patch.AppScalingMultiplier = 0 THEN
	_MatchLog^.Error("Get u8gTTC48XSVersion_PatchRawValue", "Division by Zero!");
	RETURN;
End_IF

u8gTTC48XSVersion_PatchRawValue := TO_USINT((u8gTTC48XSVersion_Patch.Value - u8gTTC48XSVersion_Patch.AppScalingOffset) * u8gTTC48XSVersion_Patch.AppScalingDivisor / u8gTTC48XSVersion_Patch.AppScalingMultiplier);

                  
END_GET
END_PROPERTY

PROPERTY u8gTTC48XSVersion_CustomRawValue : USINT
GET
                    IF u8gTTC48XSVersion_Custom.AppScalingMultiplier = 0 THEN
	_MatchLog^.Error("Get u8gTTC48XSVersion_CustomRawValue", "Division by Zero!");
	RETURN;
End_IF

u8gTTC48XSVersion_CustomRawValue := TO_USINT((u8gTTC48XSVersion_Custom.Value - u8gTTC48XSVersion_Custom.AppScalingOffset) * u8gTTC48XSVersion_Custom.AppScalingDivisor / u8gTTC48XSVersion_Custom.AppScalingMultiplier);

                  
END_GET
END_PROPERTY

PROPERTY u8gTTC510Version_MajorToolValue : USINT
GET
                    IF u8gTTC510Version_Major.ToolScalingDivisor = 0 OR u8gTTC510Version_Major.AppScalingMultiplier = 0 THEN
	_MatchLog^.Error("Get u8gTTC510Version_MajorToolValue", "Division by Zero!");
	RETURN;
END_IF

u8gTTC510Version_MajorToolValue := TO_USINT(((u8gTTC510Version_Major.Value - u8gTTC510Version_Major.AppScalingOffset) * u8gTTC510Version_Major.AppScalingDivisor / u8gTTC510Version_Major.AppScalingMultiplier * u8gTTC510Version_Major.ToolScalingMultiplier / u8gTTC510Version_Major.ToolScalingDivisor) + u8gTTC510Version_Major.ToolScalingOffset);

                  
END_GET
END_PROPERTY

PROPERTY u8gTTC510Version_MinorToolValue : USINT
GET
                    IF u8gTTC510Version_Minor.ToolScalingDivisor = 0 OR u8gTTC510Version_Minor.AppScalingMultiplier = 0 THEN
	_MatchLog^.Error("Get u8gTTC510Version_MinorToolValue", "Division by Zero!");
	RETURN;
END_IF

u8gTTC510Version_MinorToolValue := TO_USINT(((u8gTTC510Version_Minor.Value - u8gTTC510Version_Minor.AppScalingOffset) * u8gTTC510Version_Minor.AppScalingDivisor / u8gTTC510Version_Minor.AppScalingMultiplier * u8gTTC510Version_Minor.ToolScalingMultiplier / u8gTTC510Version_Minor.ToolScalingDivisor) + u8gTTC510Version_Minor.ToolScalingOffset);

                  
END_GET
END_PROPERTY

PROPERTY u8gTTC510Version_PatchToolValue : USINT
GET
                    IF u8gTTC510Version_Patch.ToolScalingDivisor = 0 OR u8gTTC510Version_Patch.AppScalingMultiplier = 0 THEN
	_MatchLog^.Error("Get u8gTTC510Version_PatchToolValue", "Division by Zero!");
	RETURN;
END_IF

u8gTTC510Version_PatchToolValue := TO_USINT(((u8gTTC510Version_Patch.Value - u8gTTC510Version_Patch.AppScalingOffset) * u8gTTC510Version_Patch.AppScalingDivisor / u8gTTC510Version_Patch.AppScalingMultiplier * u8gTTC510Version_Patch.ToolScalingMultiplier / u8gTTC510Version_Patch.ToolScalingDivisor) + u8gTTC510Version_Patch.ToolScalingOffset);

                  
END_GET
END_PROPERTY

PROPERTY u8gTTC510Version_CustomToolValue : USINT
GET
                    IF u8gTTC510Version_Custom.ToolScalingDivisor = 0 OR u8gTTC510Version_Custom.AppScalingMultiplier = 0 THEN
	_MatchLog^.Error("Get u8gTTC510Version_CustomToolValue", "Division by Zero!");
	RETURN;
END_IF

u8gTTC510Version_CustomToolValue := TO_USINT(((u8gTTC510Version_Custom.Value - u8gTTC510Version_Custom.AppScalingOffset) * u8gTTC510Version_Custom.AppScalingDivisor / u8gTTC510Version_Custom.AppScalingMultiplier * u8gTTC510Version_Custom.ToolScalingMultiplier / u8gTTC510Version_Custom.ToolScalingDivisor) + u8gTTC510Version_Custom.ToolScalingOffset);

                  
END_GET
END_PROPERTY

PROPERTY u8gTTC48XSVersion_MajorToolValue : USINT
GET
                    IF u8gTTC48XSVersion_Major.ToolScalingDivisor = 0 OR u8gTTC48XSVersion_Major.AppScalingMultiplier = 0 THEN
	_MatchLog^.Error("Get u8gTTC48XSVersion_MajorToolValue", "Division by Zero!");
	RETURN;
END_IF

u8gTTC48XSVersion_MajorToolValue := TO_USINT(((u8gTTC48XSVersion_Major.Value - u8gTTC48XSVersion_Major.AppScalingOffset) * u8gTTC48XSVersion_Major.AppScalingDivisor / u8gTTC48XSVersion_Major.AppScalingMultiplier * u8gTTC48XSVersion_Major.ToolScalingMultiplier / u8gTTC48XSVersion_Major.ToolScalingDivisor) + u8gTTC48XSVersion_Major.ToolScalingOffset);

                  
END_GET
END_PROPERTY

PROPERTY u8gTTC48XSVersion_MinorToolValue : USINT
GET
                    IF u8gTTC48XSVersion_Minor.ToolScalingDivisor = 0 OR u8gTTC48XSVersion_Minor.AppScalingMultiplier = 0 THEN
	_MatchLog^.Error("Get u8gTTC48XSVersion_MinorToolValue", "Division by Zero!");
	RETURN;
END_IF

u8gTTC48XSVersion_MinorToolValue := TO_USINT(((u8gTTC48XSVersion_Minor.Value - u8gTTC48XSVersion_Minor.AppScalingOffset) * u8gTTC48XSVersion_Minor.AppScalingDivisor / u8gTTC48XSVersion_Minor.AppScalingMultiplier * u8gTTC48XSVersion_Minor.ToolScalingMultiplier / u8gTTC48XSVersion_Minor.ToolScalingDivisor) + u8gTTC48XSVersion_Minor.ToolScalingOffset);

                  
END_GET
END_PROPERTY

PROPERTY u8gTTC48XSVersion_PatchToolValue : USINT
GET
                    IF u8gTTC48XSVersion_Patch.ToolScalingDivisor = 0 OR u8gTTC48XSVersion_Patch.AppScalingMultiplier = 0 THEN
	_MatchLog^.Error("Get u8gTTC48XSVersion_PatchToolValue", "Division by Zero!");
	RETURN;
END_IF

u8gTTC48XSVersion_PatchToolValue := TO_USINT(((u8gTTC48XSVersion_Patch.Value - u8gTTC48XSVersion_Patch.AppScalingOffset) * u8gTTC48XSVersion_Patch.AppScalingDivisor / u8gTTC48XSVersion_Patch.AppScalingMultiplier * u8gTTC48XSVersion_Patch.ToolScalingMultiplier / u8gTTC48XSVersion_Patch.ToolScalingDivisor) + u8gTTC48XSVersion_Patch.ToolScalingOffset);

                  
END_GET
END_PROPERTY

PROPERTY u8gTTC48XSVersion_CustomToolValue : USINT
GET
                    IF u8gTTC48XSVersion_Custom.ToolScalingDivisor = 0 OR u8gTTC48XSVersion_Custom.AppScalingMultiplier = 0 THEN
	_MatchLog^.Error("Get u8gTTC48XSVersion_CustomToolValue", "Division by Zero!");
	RETURN;
END_IF

u8gTTC48XSVersion_CustomToolValue := TO_USINT(((u8gTTC48XSVersion_Custom.Value - u8gTTC48XSVersion_Custom.AppScalingOffset) * u8gTTC48XSVersion_Custom.AppScalingDivisor / u8gTTC48XSVersion_Custom.AppScalingMultiplier * u8gTTC48XSVersion_Custom.ToolScalingMultiplier / u8gTTC48XSVersion_Custom.ToolScalingDivisor) + u8gTTC48XSVersion_Custom.ToolScalingOffset);

                  
END_GET
END_PROPERTY

METHOD InitializeCanSignals
                  u8gTTC510Version_Major.AppScalingDivisor :=1;
u8gTTC510Version_Major.AppScalingMultiplier :=1;
u8gTTC510Version_Major.AppScalingOffset :=0;
u8gTTC510Version_Major.AppUnit :="";
u8gTTC510Version_Major.CanDefault :=0;
u8gTTC510Version_Major.CanInit :=0;
u8gTTC510Version_Major.CanMax :=VBasic.LibConst.U8_MAX;
u8gTTC510Version_Major.CanMin :=VBasic.LibConst.U8_MIN;
u8gTTC510Version_Major.CanUnit :="";
u8gTTC510Version_Major.Description :="Program Version Major C1 TTC510";
u8gTTC510Version_Major.ErrorReaction := eErrorReaction.ERSIG_DFLT;
u8gTTC510Version_Major.ReceiverAdress :=1;
u8gTTC510Version_Major.ToolScalingDivisor :=1;
u8gTTC510Version_Major.ToolScalingMultiplier :=1;
u8gTTC510Version_Major.ToolScalingOffset :=0;
u8gTTC510Version_Major.ToolUnit :="";

u8gTTC510Version_Minor.AppScalingDivisor :=1;
u8gTTC510Version_Minor.AppScalingMultiplier :=1;
u8gTTC510Version_Minor.AppScalingOffset :=0;
u8gTTC510Version_Minor.AppUnit :="";
u8gTTC510Version_Minor.CanDefault :=0;
u8gTTC510Version_Minor.CanInit :=0;
u8gTTC510Version_Minor.CanMax :=VBasic.LibConst.U8_MAX;
u8gTTC510Version_Minor.CanMin :=VBasic.LibConst.U8_MIN;
u8gTTC510Version_Minor.CanUnit :="";
u8gTTC510Version_Minor.Description :="Program Version Minor C1 TTC510";
u8gTTC510Version_Minor.ErrorReaction := eErrorReaction.ERSIG_DFLT;
u8gTTC510Version_Minor.ReceiverAdress :=1;
u8gTTC510Version_Minor.ToolScalingDivisor :=1;
u8gTTC510Version_Minor.ToolScalingMultiplier :=1;
u8gTTC510Version_Minor.ToolScalingOffset :=0;
u8gTTC510Version_Minor.ToolUnit :="";

u8gTTC510Version_Patch.AppScalingDivisor :=1;
u8gTTC510Version_Patch.AppScalingMultiplier :=1;
u8gTTC510Version_Patch.AppScalingOffset :=0;
u8gTTC510Version_Patch.AppUnit :="";
u8gTTC510Version_Patch.CanDefault :=0;
u8gTTC510Version_Patch.CanInit :=0;
u8gTTC510Version_Patch.CanMax :=VBasic.LibConst.U8_MAX;
u8gTTC510Version_Patch.CanMin :=VBasic.LibConst.U8_MIN;
u8gTTC510Version_Patch.CanUnit :="";
u8gTTC510Version_Patch.Description :="Program Version Patch C1 TTC510";
u8gTTC510Version_Patch.ErrorReaction := eErrorReaction.ERSIG_DFLT;
u8gTTC510Version_Patch.ReceiverAdress :=1;
u8gTTC510Version_Patch.ToolScalingDivisor :=1;
u8gTTC510Version_Patch.ToolScalingMultiplier :=1;
u8gTTC510Version_Patch.ToolScalingOffset :=0;
u8gTTC510Version_Patch.ToolUnit :="";

u8gTTC510Version_Custom.AppScalingDivisor :=1;
u8gTTC510Version_Custom.AppScalingMultiplier :=1;
u8gTTC510Version_Custom.AppScalingOffset :=0;
u8gTTC510Version_Custom.AppUnit :="";
u8gTTC510Version_Custom.CanDefault :=0;
u8gTTC510Version_Custom.CanInit :=0;
u8gTTC510Version_Custom.CanMax :=VBasic.LibConst.U8_MAX;
u8gTTC510Version_Custom.CanMin :=VBasic.LibConst.U8_MIN;
u8gTTC510Version_Custom.CanUnit :="";
u8gTTC510Version_Custom.Description :="Program Version Custom C1 TTC510";
u8gTTC510Version_Custom.ErrorReaction := eErrorReaction.ERSIG_DFLT;
u8gTTC510Version_Custom.ReceiverAdress :=1;
u8gTTC510Version_Custom.ToolScalingDivisor :=1;
u8gTTC510Version_Custom.ToolScalingMultiplier :=1;
u8gTTC510Version_Custom.ToolScalingOffset :=0;
u8gTTC510Version_Custom.ToolUnit :="";

u8gTTC48XSVersion_Major.AppScalingDivisor :=1;
u8gTTC48XSVersion_Major.AppScalingMultiplier :=1;
u8gTTC48XSVersion_Major.AppScalingOffset :=0;
u8gTTC48XSVersion_Major.AppUnit :="";
u8gTTC48XSVersion_Major.CanDefault :=0;
u8gTTC48XSVersion_Major.CanInit :=0;
u8gTTC48XSVersion_Major.CanMax :=VBasic.LibConst.U8_MAX;
u8gTTC48XSVersion_Major.CanMin :=VBasic.LibConst.U8_MIN;
u8gTTC48XSVersion_Major.CanUnit :="";
u8gTTC48XSVersion_Major.Description :="Program Version Major TTC48XS";
u8gTTC48XSVersion_Major.ErrorReaction := eErrorReaction.ERSIG_DFLT;
u8gTTC48XSVersion_Major.ReceiverAdress :=1;
u8gTTC48XSVersion_Major.ToolScalingDivisor :=1;
u8gTTC48XSVersion_Major.ToolScalingMultiplier :=1;
u8gTTC48XSVersion_Major.ToolScalingOffset :=0;
u8gTTC48XSVersion_Major.ToolUnit :="";

u8gTTC48XSVersion_Minor.AppScalingDivisor :=1;
u8gTTC48XSVersion_Minor.AppScalingMultiplier :=1;
u8gTTC48XSVersion_Minor.AppScalingOffset :=0;
u8gTTC48XSVersion_Minor.AppUnit :="";
u8gTTC48XSVersion_Minor.CanDefault :=0;
u8gTTC48XSVersion_Minor.CanInit :=0;
u8gTTC48XSVersion_Minor.CanMax :=VBasic.LibConst.U8_MAX;
u8gTTC48XSVersion_Minor.CanMin :=VBasic.LibConst.U8_MIN;
u8gTTC48XSVersion_Minor.CanUnit :="";
u8gTTC48XSVersion_Minor.Description :="Program Version Minor TTC48XS";
u8gTTC48XSVersion_Minor.ErrorReaction := eErrorReaction.ERSIG_DFLT;
u8gTTC48XSVersion_Minor.ReceiverAdress :=1;
u8gTTC48XSVersion_Minor.ToolScalingDivisor :=1;
u8gTTC48XSVersion_Minor.ToolScalingMultiplier :=1;
u8gTTC48XSVersion_Minor.ToolScalingOffset :=0;
u8gTTC48XSVersion_Minor.ToolUnit :="";

u8gTTC48XSVersion_Patch.AppScalingDivisor :=1;
u8gTTC48XSVersion_Patch.AppScalingMultiplier :=1;
u8gTTC48XSVersion_Patch.AppScalingOffset :=0;
u8gTTC48XSVersion_Patch.AppUnit :="";
u8gTTC48XSVersion_Patch.CanDefault :=0;
u8gTTC48XSVersion_Patch.CanInit :=0;
u8gTTC48XSVersion_Patch.CanMax :=VBasic.LibConst.U8_MAX;
u8gTTC48XSVersion_Patch.CanMin :=VBasic.LibConst.U8_MIN;
u8gTTC48XSVersion_Patch.CanUnit :="";
u8gTTC48XSVersion_Patch.Description :="Program Version Patch TTC48XS";
u8gTTC48XSVersion_Patch.ErrorReaction := eErrorReaction.ERSIG_DFLT;
u8gTTC48XSVersion_Patch.ReceiverAdress :=1;
u8gTTC48XSVersion_Patch.ToolScalingDivisor :=1;
u8gTTC48XSVersion_Patch.ToolScalingMultiplier :=1;
u8gTTC48XSVersion_Patch.ToolScalingOffset :=0;
u8gTTC48XSVersion_Patch.ToolUnit :="";

u8gTTC48XSVersion_Custom.AppScalingDivisor :=1;
u8gTTC48XSVersion_Custom.AppScalingMultiplier :=1;
u8gTTC48XSVersion_Custom.AppScalingOffset :=0;
u8gTTC48XSVersion_Custom.AppUnit :="";
u8gTTC48XSVersion_Custom.CanDefault :=0;
u8gTTC48XSVersion_Custom.CanInit :=0;
u8gTTC48XSVersion_Custom.CanMax :=VBasic.LibConst.U8_MAX;
u8gTTC48XSVersion_Custom.CanMin :=VBasic.LibConst.U8_MIN;
u8gTTC48XSVersion_Custom.CanUnit :="";
u8gTTC48XSVersion_Custom.Description :="Program Version Custom TTC48XS";
u8gTTC48XSVersion_Custom.ErrorReaction := eErrorReaction.ERSIG_DFLT;
u8gTTC48XSVersion_Custom.ReceiverAdress :=1;
u8gTTC48XSVersion_Custom.ToolScalingDivisor :=1;
u8gTTC48XSVersion_Custom.ToolScalingMultiplier :=1;
u8gTTC48XSVersion_Custom.ToolScalingOffset :=0;
u8gTTC48XSVersion_Custom.ToolUnit :="";


                
END_METHOD
END_FUNCTION_BLOCK

FUNCTION_BLOCK Msg9C1SendToOpusMessageClass EXTENDS CanReceiveMessageClass
  VAR_INPUT
    boAutoModeActivate : BoolCanSignalClass;
    boSilenceModeActivate : BoolCanSignalClass;
    boForcingModeActivate : BoolCanSignalClass;
    boForcingRegenlow : BoolCanSignalClass;
    boForcingRegenHigh : BoolCanSignalClass;
    boAskReloadWithGenerator : BoolCanSignalClass;
    boReloadWithGeneratorOn : BoolCanSignalClass;
    boAlarmCptNbrRegenFinish : BoolCanSignalClass;
    boElectricMotorForbidden : BoolCanSignalClass;
    boPictoColdOilTankTemperature : BoolCanSignalClass;
    boRecoveryReductionRatio : BoolCanSignalClass;
    u16RemainingRegenTimeAverage : UInt16CanSignalClass;
    u16TotalRegenHours : UInt16CanSignalClass;
    Counter : UInt32CanSignalClass;
  END_VAR

            
          

METHOD SetData
  VAR_INPUT
    CanMsgPointer : POINTER TO CanMessageClass;
  END_VAR
                  IF IsValidPointer(canMsgPointer,'SetData') THEN
	SUPER^.SetData(CanMsgPointer);
	//Set the new data
	boAutoModeActivate.Value := canMsgPointer^.GetBoolOnBit(0);
	boSilenceModeActivate.Value := canMsgPointer^.GetBoolOnBit(1);
	boForcingModeActivate.Value := canMsgPointer^.GetBoolOnBit(2);
	boForcingRegenlow.Value := canMsgPointer^.GetBoolOnBit(3);
	boForcingRegenHigh.Value := canMsgPointer^.GetBoolOnBit(4);
	boAskReloadWithGenerator.Value := canMsgPointer^.GetBoolOnBit(5);
	boReloadWithGeneratorOn.Value := canMsgPointer^.GetBoolOnBit(6);
	boAlarmCptNbrRegenFinish.Value := canMsgPointer^.GetBoolOnBit(7);
	boElectricMotorForbidden.Value := canMsgPointer^.GetBoolOnBit(8);
	boPictoColdOilTankTemperature.Value := canMsgPointer^.GetBoolOnBit(9);
	boRecoveryReductionRatio.Value := canMsgPointer^.GetBoolOnBit(10);
	u16RemainingRegenTimeAverage.Value := canMsgPointer^.GetUint16(16);
	u16TotalRegenHours.Value := canMsgPointer^.GetUint16(32);
	//And increase the counter
	Counter.Value := CanMsgPointer^.Counter.Value;
END_IF

                
END_METHOD

PROPERTY boAutoModeActivateRawValue : BOOL
GET
                    boAutoModeActivateRawValue := boAutoModeActivate.Value;

                  
END_GET
END_PROPERTY

PROPERTY boSilenceModeActivateRawValue : BOOL
GET
                    boSilenceModeActivateRawValue := boSilenceModeActivate.Value;

                  
END_GET
END_PROPERTY

PROPERTY boForcingModeActivateRawValue : BOOL
GET
                    boForcingModeActivateRawValue := boForcingModeActivate.Value;

                  
END_GET
END_PROPERTY

PROPERTY boForcingRegenlowRawValue : BOOL
GET
                    boForcingRegenlowRawValue := boForcingRegenlow.Value;

                  
END_GET
END_PROPERTY

PROPERTY boForcingRegenHighRawValue : BOOL
GET
                    boForcingRegenHighRawValue := boForcingRegenHigh.Value;

                  
END_GET
END_PROPERTY

PROPERTY boAskReloadWithGeneratorRawValue : BOOL
GET
                    boAskReloadWithGeneratorRawValue := boAskReloadWithGenerator.Value;

                  
END_GET
END_PROPERTY

PROPERTY boReloadWithGeneratorOnRawValue : BOOL
GET
                    boReloadWithGeneratorOnRawValue := boReloadWithGeneratorOn.Value;

                  
END_GET
END_PROPERTY

PROPERTY boAlarmCptNbrRegenFinishRawValue : BOOL
GET
                    boAlarmCptNbrRegenFinishRawValue := boAlarmCptNbrRegenFinish.Value;

                  
END_GET
END_PROPERTY

PROPERTY boElectricMotorForbiddenRawValue : BOOL
GET
                    boElectricMotorForbiddenRawValue := boElectricMotorForbidden.Value;

                  
END_GET
END_PROPERTY

PROPERTY boPictoColdOilTankTemperatureRawValue : BOOL
GET
                    boPictoColdOilTankTemperatureRawValue := boPictoColdOilTankTemperature.Value;

                  
END_GET
END_PROPERTY

PROPERTY boRecoveryReductionRatioRawValue : BOOL
GET
                    boRecoveryReductionRatioRawValue := boRecoveryReductionRatio.Value;

                  
END_GET
END_PROPERTY

PROPERTY u16RemainingRegenTimeAverageRawValue : UINT
GET
                    IF u16RemainingRegenTimeAverage.AppScalingMultiplier = 0 THEN
	_MatchLog^.Error("Get u16RemainingRegenTimeAverageRawValue", "Division by Zero!");
	RETURN;
End_IF

u16RemainingRegenTimeAverageRawValue := TO_UINT((u16RemainingRegenTimeAverage.Value - u16RemainingRegenTimeAverage.AppScalingOffset) * u16RemainingRegenTimeAverage.AppScalingDivisor / u16RemainingRegenTimeAverage.AppScalingMultiplier);

                  
END_GET
END_PROPERTY

PROPERTY u16TotalRegenHoursRawValue : UINT
GET
                    IF u16TotalRegenHours.AppScalingMultiplier = 0 THEN
	_MatchLog^.Error("Get u16TotalRegenHoursRawValue", "Division by Zero!");
	RETURN;
End_IF

u16TotalRegenHoursRawValue := TO_UINT((u16TotalRegenHours.Value - u16TotalRegenHours.AppScalingOffset) * u16TotalRegenHours.AppScalingDivisor / u16TotalRegenHours.AppScalingMultiplier);

                  
END_GET
END_PROPERTY

PROPERTY boAutoModeActivateToolValue : BOOL
GET
                    boAutoModeActivateToolValue := boAutoModeActivate.Value;

                  
END_GET
END_PROPERTY

PROPERTY boSilenceModeActivateToolValue : BOOL
GET
                    boSilenceModeActivateToolValue := boSilenceModeActivate.Value;

                  
END_GET
END_PROPERTY

PROPERTY boForcingModeActivateToolValue : BOOL
GET
                    boForcingModeActivateToolValue := boForcingModeActivate.Value;

                  
END_GET
END_PROPERTY

PROPERTY boForcingRegenlowToolValue : BOOL
GET
                    boForcingRegenlowToolValue := boForcingRegenlow.Value;

                  
END_GET
END_PROPERTY

PROPERTY boForcingRegenHighToolValue : BOOL
GET
                    boForcingRegenHighToolValue := boForcingRegenHigh.Value;

                  
END_GET
END_PROPERTY

PROPERTY boAskReloadWithGeneratorToolValue : BOOL
GET
                    boAskReloadWithGeneratorToolValue := boAskReloadWithGenerator.Value;

                  
END_GET
END_PROPERTY

PROPERTY boReloadWithGeneratorOnToolValue : BOOL
GET
                    boReloadWithGeneratorOnToolValue := boReloadWithGeneratorOn.Value;

                  
END_GET
END_PROPERTY

PROPERTY boAlarmCptNbrRegenFinishToolValue : BOOL
GET
                    boAlarmCptNbrRegenFinishToolValue := boAlarmCptNbrRegenFinish.Value;

                  
END_GET
END_PROPERTY

PROPERTY boElectricMotorForbiddenToolValue : BOOL
GET
                    boElectricMotorForbiddenToolValue := boElectricMotorForbidden.Value;

                  
END_GET
END_PROPERTY

PROPERTY boPictoColdOilTankTemperatureToolValue : BOOL
GET
                    boPictoColdOilTankTemperatureToolValue := boPictoColdOilTankTemperature.Value;

                  
END_GET
END_PROPERTY

PROPERTY boRecoveryReductionRatioToolValue : BOOL
GET
                    boRecoveryReductionRatioToolValue := boRecoveryReductionRatio.Value;

                  
END_GET
END_PROPERTY

PROPERTY u16RemainingRegenTimeAverageToolValue : UINT
GET
                    IF u16RemainingRegenTimeAverage.ToolScalingDivisor = 0 OR u16RemainingRegenTimeAverage.AppScalingMultiplier = 0 THEN
	_MatchLog^.Error("Get u16RemainingRegenTimeAverageToolValue", "Division by Zero!");
	RETURN;
END_IF

u16RemainingRegenTimeAverageToolValue := TO_UINT(((u16RemainingRegenTimeAverage.Value - u16RemainingRegenTimeAverage.AppScalingOffset) * u16RemainingRegenTimeAverage.AppScalingDivisor / u16RemainingRegenTimeAverage.AppScalingMultiplier * u16RemainingRegenTimeAverage.ToolScalingMultiplier / u16RemainingRegenTimeAverage.ToolScalingDivisor) + u16RemainingRegenTimeAverage.ToolScalingOffset);

                  
END_GET
END_PROPERTY

PROPERTY u16TotalRegenHoursToolValue : UINT
GET
                    IF u16TotalRegenHours.ToolScalingDivisor = 0 OR u16TotalRegenHours.AppScalingMultiplier = 0 THEN
	_MatchLog^.Error("Get u16TotalRegenHoursToolValue", "Division by Zero!");
	RETURN;
END_IF

u16TotalRegenHoursToolValue := TO_UINT(((u16TotalRegenHours.Value - u16TotalRegenHours.AppScalingOffset) * u16TotalRegenHours.AppScalingDivisor / u16TotalRegenHours.AppScalingMultiplier * u16TotalRegenHours.ToolScalingMultiplier / u16TotalRegenHours.ToolScalingDivisor) + u16TotalRegenHours.ToolScalingOffset);

                  
END_GET
END_PROPERTY

METHOD InitializeCanSignals
                  boAutoModeActivate.AppScalingDivisor :=1;
boAutoModeActivate.AppScalingMultiplier :=1;
boAutoModeActivate.AppScalingOffset :=0;
boAutoModeActivate.AppUnit :="";
boAutoModeActivate.CanDefault :=0;
boAutoModeActivate.CanInit :=0;
boAutoModeActivate.CanMax :=1;
boAutoModeActivate.CanMin :=0;
boAutoModeActivate.CanUnit :="";
boAutoModeActivate.Description :="new signal";
boAutoModeActivate.ErrorReaction := eErrorReaction.ERSIG_DFLT;
boAutoModeActivate.ReceiverAdress :=1;
boAutoModeActivate.ToolScalingDivisor :=1;
boAutoModeActivate.ToolScalingMultiplier :=1;
boAutoModeActivate.ToolScalingOffset :=0;
boAutoModeActivate.ToolUnit :="";

boSilenceModeActivate.AppScalingDivisor :=1;
boSilenceModeActivate.AppScalingMultiplier :=1;
boSilenceModeActivate.AppScalingOffset :=0;
boSilenceModeActivate.AppUnit :="";
boSilenceModeActivate.CanDefault :=0;
boSilenceModeActivate.CanInit :=0;
boSilenceModeActivate.CanMax :=1;
boSilenceModeActivate.CanMin :=0;
boSilenceModeActivate.CanUnit :="";
boSilenceModeActivate.Description :="new signal";
boSilenceModeActivate.ErrorReaction := eErrorReaction.ERSIG_DFLT;
boSilenceModeActivate.ReceiverAdress :=1;
boSilenceModeActivate.ToolScalingDivisor :=1;
boSilenceModeActivate.ToolScalingMultiplier :=1;
boSilenceModeActivate.ToolScalingOffset :=0;
boSilenceModeActivate.ToolUnit :="";

boForcingModeActivate.AppScalingDivisor :=1;
boForcingModeActivate.AppScalingMultiplier :=1;
boForcingModeActivate.AppScalingOffset :=0;
boForcingModeActivate.AppUnit :="";
boForcingModeActivate.CanDefault :=0;
boForcingModeActivate.CanInit :=0;
boForcingModeActivate.CanMax :=1;
boForcingModeActivate.CanMin :=0;
boForcingModeActivate.CanUnit :="";
boForcingModeActivate.Description :="new signal";
boForcingModeActivate.ErrorReaction := eErrorReaction.ERSIG_DFLT;
boForcingModeActivate.ReceiverAdress :=1;
boForcingModeActivate.ToolScalingDivisor :=1;
boForcingModeActivate.ToolScalingMultiplier :=1;
boForcingModeActivate.ToolScalingOffset :=0;
boForcingModeActivate.ToolUnit :="";

boForcingRegenlow.AppScalingDivisor :=1;
boForcingRegenlow.AppScalingMultiplier :=1;
boForcingRegenlow.AppScalingOffset :=0;
boForcingRegenlow.AppUnit :="";
boForcingRegenlow.CanDefault :=0;
boForcingRegenlow.CanInit :=0;
boForcingRegenlow.CanMax :=1;
boForcingRegenlow.CanMin :=0;
boForcingRegenlow.CanUnit :="";
boForcingRegenlow.Description :="new signal";
boForcingRegenlow.ErrorReaction := eErrorReaction.ERSIG_DFLT;
boForcingRegenlow.ReceiverAdress :=1;
boForcingRegenlow.ToolScalingDivisor :=1;
boForcingRegenlow.ToolScalingMultiplier :=1;
boForcingRegenlow.ToolScalingOffset :=0;
boForcingRegenlow.ToolUnit :="";

boForcingRegenHigh.AppScalingDivisor :=1;
boForcingRegenHigh.AppScalingMultiplier :=1;
boForcingRegenHigh.AppScalingOffset :=0;
boForcingRegenHigh.AppUnit :="";
boForcingRegenHigh.CanDefault :=0;
boForcingRegenHigh.CanInit :=0;
boForcingRegenHigh.CanMax :=1;
boForcingRegenHigh.CanMin :=0;
boForcingRegenHigh.CanUnit :="";
boForcingRegenHigh.Description :="new signal";
boForcingRegenHigh.ErrorReaction := eErrorReaction.ERSIG_DFLT;
boForcingRegenHigh.ReceiverAdress :=1;
boForcingRegenHigh.ToolScalingDivisor :=1;
boForcingRegenHigh.ToolScalingMultiplier :=1;
boForcingRegenHigh.ToolScalingOffset :=0;
boForcingRegenHigh.ToolUnit :="";

boAskReloadWithGenerator.AppScalingDivisor :=1;
boAskReloadWithGenerator.AppScalingMultiplier :=1;
boAskReloadWithGenerator.AppScalingOffset :=0;
boAskReloadWithGenerator.AppUnit :="";
boAskReloadWithGenerator.CanDefault :=0;
boAskReloadWithGenerator.CanInit :=0;
boAskReloadWithGenerator.CanMax :=1;
boAskReloadWithGenerator.CanMin :=0;
boAskReloadWithGenerator.CanUnit :="";
boAskReloadWithGenerator.Description :="new signal";
boAskReloadWithGenerator.ErrorReaction := eErrorReaction.ERSIG_DFLT;
boAskReloadWithGenerator.ReceiverAdress :=1;
boAskReloadWithGenerator.ToolScalingDivisor :=1;
boAskReloadWithGenerator.ToolScalingMultiplier :=1;
boAskReloadWithGenerator.ToolScalingOffset :=0;
boAskReloadWithGenerator.ToolUnit :="";

boReloadWithGeneratorOn.AppScalingDivisor :=1;
boReloadWithGeneratorOn.AppScalingMultiplier :=1;
boReloadWithGeneratorOn.AppScalingOffset :=0;
boReloadWithGeneratorOn.AppUnit :="";
boReloadWithGeneratorOn.CanDefault :=0;
boReloadWithGeneratorOn.CanInit :=0;
boReloadWithGeneratorOn.CanMax :=1;
boReloadWithGeneratorOn.CanMin :=0;
boReloadWithGeneratorOn.CanUnit :="";
boReloadWithGeneratorOn.Description :="new signal";
boReloadWithGeneratorOn.ErrorReaction := eErrorReaction.ERSIG_DFLT;
boReloadWithGeneratorOn.ReceiverAdress :=1;
boReloadWithGeneratorOn.ToolScalingDivisor :=1;
boReloadWithGeneratorOn.ToolScalingMultiplier :=1;
boReloadWithGeneratorOn.ToolScalingOffset :=0;
boReloadWithGeneratorOn.ToolUnit :="";

boAlarmCptNbrRegenFinish.AppScalingDivisor :=1;
boAlarmCptNbrRegenFinish.AppScalingMultiplier :=1;
boAlarmCptNbrRegenFinish.AppScalingOffset :=0;
boAlarmCptNbrRegenFinish.AppUnit :="";
boAlarmCptNbrRegenFinish.CanDefault :=0;
boAlarmCptNbrRegenFinish.CanInit :=0;
boAlarmCptNbrRegenFinish.CanMax :=1;
boAlarmCptNbrRegenFinish.CanMin :=0;
boAlarmCptNbrRegenFinish.CanUnit :="";
boAlarmCptNbrRegenFinish.Description :="new signal";
boAlarmCptNbrRegenFinish.ErrorReaction := eErrorReaction.ERSIG_DFLT;
boAlarmCptNbrRegenFinish.ReceiverAdress :=1;
boAlarmCptNbrRegenFinish.ToolScalingDivisor :=1;
boAlarmCptNbrRegenFinish.ToolScalingMultiplier :=1;
boAlarmCptNbrRegenFinish.ToolScalingOffset :=0;
boAlarmCptNbrRegenFinish.ToolUnit :="";

boElectricMotorForbidden.AppScalingDivisor :=1;
boElectricMotorForbidden.AppScalingMultiplier :=1;
boElectricMotorForbidden.AppScalingOffset :=0;
boElectricMotorForbidden.AppUnit :="";
boElectricMotorForbidden.CanDefault :=0;
boElectricMotorForbidden.CanInit :=0;
boElectricMotorForbidden.CanMax :=1;
boElectricMotorForbidden.CanMin :=0;
boElectricMotorForbidden.CanUnit :="";
boElectricMotorForbidden.Description :="new signal";
boElectricMotorForbidden.ErrorReaction := eErrorReaction.ERSIG_DFLT;
boElectricMotorForbidden.ReceiverAdress :=1;
boElectricMotorForbidden.ToolScalingDivisor :=1;
boElectricMotorForbidden.ToolScalingMultiplier :=1;
boElectricMotorForbidden.ToolScalingOffset :=0;
boElectricMotorForbidden.ToolUnit :="";

boPictoColdOilTankTemperature.AppScalingDivisor :=1;
boPictoColdOilTankTemperature.AppScalingMultiplier :=1;
boPictoColdOilTankTemperature.AppScalingOffset :=0;
boPictoColdOilTankTemperature.AppUnit :="";
boPictoColdOilTankTemperature.CanDefault :=0;
boPictoColdOilTankTemperature.CanInit :=0;
boPictoColdOilTankTemperature.CanMax :=1;
boPictoColdOilTankTemperature.CanMin :=0;
boPictoColdOilTankTemperature.CanUnit :="";
boPictoColdOilTankTemperature.Description :="new signal";
boPictoColdOilTankTemperature.ErrorReaction := eErrorReaction.ERSIG_DFLT;
boPictoColdOilTankTemperature.ReceiverAdress :=1;
boPictoColdOilTankTemperature.ToolScalingDivisor :=1;
boPictoColdOilTankTemperature.ToolScalingMultiplier :=1;
boPictoColdOilTankTemperature.ToolScalingOffset :=0;
boPictoColdOilTankTemperature.ToolUnit :="";

boRecoveryReductionRatio.AppScalingDivisor :=1;
boRecoveryReductionRatio.AppScalingMultiplier :=1;
boRecoveryReductionRatio.AppScalingOffset :=0;
boRecoveryReductionRatio.AppUnit :="";
boRecoveryReductionRatio.CanDefault :=0;
boRecoveryReductionRatio.CanInit :=0;
boRecoveryReductionRatio.CanMax :=1;
boRecoveryReductionRatio.CanMin :=0;
boRecoveryReductionRatio.CanUnit :="";
boRecoveryReductionRatio.Description :="new signal";
boRecoveryReductionRatio.ErrorReaction := eErrorReaction.ERSIG_DFLT;
boRecoveryReductionRatio.ReceiverAdress :=1;
boRecoveryReductionRatio.ToolScalingDivisor :=1;
boRecoveryReductionRatio.ToolScalingMultiplier :=1;
boRecoveryReductionRatio.ToolScalingOffset :=0;
boRecoveryReductionRatio.ToolUnit :="";

u16RemainingRegenTimeAverage.AppScalingDivisor :=1;
u16RemainingRegenTimeAverage.AppScalingMultiplier :=1;
u16RemainingRegenTimeAverage.AppScalingOffset :=0;
u16RemainingRegenTimeAverage.AppUnit :="";
u16RemainingRegenTimeAverage.CanDefault :=0;
u16RemainingRegenTimeAverage.CanInit :=0;
u16RemainingRegenTimeAverage.CanMax :=VBasic.LibConst.U16_MAX;
u16RemainingRegenTimeAverage.CanMin :=VBasic.LibConst.U16_MIN;
u16RemainingRegenTimeAverage.CanUnit :="";
u16RemainingRegenTimeAverage.Description :="new signal";
u16RemainingRegenTimeAverage.ErrorReaction := eErrorReaction.ERSIG_DFLT;
u16RemainingRegenTimeAverage.ReceiverAdress :=1;
u16RemainingRegenTimeAverage.ToolScalingDivisor :=1;
u16RemainingRegenTimeAverage.ToolScalingMultiplier :=1;
u16RemainingRegenTimeAverage.ToolScalingOffset :=0;
u16RemainingRegenTimeAverage.ToolUnit :="";

u16TotalRegenHours.AppScalingDivisor :=1;
u16TotalRegenHours.AppScalingMultiplier :=1;
u16TotalRegenHours.AppScalingOffset :=0;
u16TotalRegenHours.AppUnit :="";
u16TotalRegenHours.CanDefault :=0;
u16TotalRegenHours.CanInit :=0;
u16TotalRegenHours.CanMax :=VBasic.LibConst.U16_MAX;
u16TotalRegenHours.CanMin :=VBasic.LibConst.U16_MIN;
u16TotalRegenHours.CanUnit :="";
u16TotalRegenHours.Description :="new signal";
u16TotalRegenHours.ErrorReaction := eErrorReaction.ERSIG_DFLT;
u16TotalRegenHours.ReceiverAdress :=1;
u16TotalRegenHours.ToolScalingDivisor :=1;
u16TotalRegenHours.ToolScalingMultiplier :=1;
u16TotalRegenHours.ToolScalingOffset :=0;
u16TotalRegenHours.ToolUnit :="";


                
END_METHOD
END_FUNCTION_BLOCK

FUNCTION MatchLibInit_Addresses : BOOL

            // **********************************************************************************************************************
// *  AUTO-GENERATED:  PdtCodeBuilder.dll (Version: 1.2.7, Build: 080)
// *  Itf-Version:     1.7.0
// *  Pdt-Version:     2.11.72.172
// *  Pdt-ProjVersion: 0.0.0
// *  Match-Version:   07.04.00.00
// *  Copyright (C) 2012 HYDAC SYSTEM GMBH -  All rights reserved.
// *  Entwicklungsbüro Berlin - Zum Kiesberg 16 - D-14979 Großbeeren
// *  2025-04-18 16:40:50 created
// **********************************************************************************************************************


gLib_MatchInitializer.ControllerCount := 0;
gLib_MatchInitializer.DisplaySA := 16#2F;
MatchVars.J1939_SA_MST := 16#E8; // Source Address servicetool (BYTE)
MatchVars.J1939_SA_TCP := 16#2E; // Source Address servicetool TCP (BYTE)
gLib_MatchInitializer.ControllerSA[gLib_MatchInitializer.ControllerCount] := 16#20;
gLib_MatchInitializer.ControllerSymbols[gLib_MatchInitializer.ControllerCount] := "C0";
gLib_MatchInitializer.ControllerCount := gLib_MatchInitializer.ControllerCount + 1;
gLib_MatchInitializer.ControllerSA[gLib_MatchInitializer.ControllerCount] := 16#21;
gLib_MatchInitializer.ControllerSymbols[gLib_MatchInitializer.ControllerCount] := "C1";
gLib_MatchInitializer.ControllerCount := gLib_MatchInitializer.ControllerCount + 1;

          
END_FUNCTION

FUNCTION MatchLibInit_VersionInformation : BOOL

            gLib_MatchInitializer.VersionInformation.EcuNumber.Value := '2';
gLib_MatchInitializer.VersionInformation.EcuNumber.CompanyCode := 'HY1234HY';
gLib_MatchInitializer.VersionInformation.MstProjectIdentifier.IdCompanyCode := "HY1234HY";
gLib_MatchInitializer.VersionInformation.MstProjectIdentifier.IdMachineName := "Skyrailer";
gLib_MatchInitializer.VersionInformation.MstProjectIdentifier.IdGuid := "DemoMachine_HY1234HY_18264adf-9280-4e7b-a965-67acf0df2d1c";
gLib_MatchInitializer.VersionInformation.VehicleIdA.Brand := '-';
gLib_MatchInitializer.VersionInformation.VehicleIdA.Manufacturer := 'Neotec skyrailer';
gLib_MatchInitializer.VersionInformation.VehicleIdA.ManufacturerLocation := '-';
gLib_MatchInitializer.VersionInformation.VehicleIdA.MachineType := 'Nacelle';
gLib_MatchInitializer.VersionInformation.VehicleIdA.PartNumber := '-';
gLib_MatchInitializer.VersionInformation.VehicleIdA.SalesName := 'Skyrailer';
gLib_MatchInitializer.VersionInformation.ApplicationSoftware.Major := '0';
gLib_MatchInitializer.VersionInformation.ApplicationSoftware.Minor := '0';
gLib_MatchInitializer.VersionInformation.ApplicationSoftware.Index := '0';
gLib_MatchInitializer.VersionInformation.ApplicationSoftware.DevStep := '623';
gLib_MatchInitializer.VersionInformation.ApplicationSoftware.CDate := '18.04.2025';
gLib_MatchInitializer.VersionInformation.ApplicationSoftware.CTime := '16:40:32';
gLib_MatchInitializer.VersionInformation.EcuHardware.VersionNumber := '-';
gLib_MatchInitializer.VersionInformation.EcuHardware.ControllerType := 'EVISION2';
gLib_MatchInitializer.VersionInformation.Compiler.Supplier := '3S';
gLib_MatchInitializer.VersionInformation.Compiler.Version := '-';
gLib_MatchInitializer.VersionInformation.Compiler.BuildProcNumber := '-';

          
END_FUNCTION
